PROGRAM MAIN
VAR
	linearNC : LinearServoNC;
	linearCLMC : LinearClearLinkMC;
	linearAP : LinearAirPiston;
	
	insertion : Insertion2D;
END_VAR

linearNC(
	bEnable:= TRUE, 
	ready=> , 
	position=> , 
	velocity=> , 
	sensorDefaultState:= TRUE, 
	homeAt0:= TRUE, 
	allowDualSideTraverse:= TRUE);
	
linearCLMC(
	bEnable:= TRUE, 
	pulse=> , 
	brakeRelease=> , 
	enable=> , 
	A=> , 
	B=> , 
	clear=> , 
	sensorDefaultState:= TRUE, 
	homeAt0:= FALSE, 
	allowDualSideTraverse:= FALSE);
	
linearAP(bEnable:= TRUE, valveExtend=> , valveRetract=> , sensorDefaultState:= FALSE);

insertion(
	slider:= linearCLMC, 
	screw:= linearNC, 
	contact=> , 
	active=> , 
	error=> , 
	home=> , 
	homingComplete=> , 
	sliderPos=> );

END_PROGRAM

(* stored: Version 1.1.0.1, ProductVersion 3.1.4024.11
   POU MAIN: Id {2da2c240-123a-4dc5-8fca-5f9b4ed2e0c6}, SpecialFunc None *)
